Staubli VAL3: oCryoShortOut.pgx

public program oCryoShortOut(num nChoice (dimensions=1))
// oCryoShortOut
begin
  dioSet(oCryoShortOut,nChoice)
end
